PROGRAM DatenRangieren
VAR	
	VersionsText: STRING := 'LAP 2010/3 Ofentuersteuerung V3.0';
END_VAR

STRNCPY (ADR( _plcToPc.PlcToPc[96]), ADR( VersionsText), SIZEOF(VersionsText));

IF _PcToPlc.PcToPlc[96] = 16#00 THEN	// lokale Ein- und Ausgänge verwenden
	
ELSE	// Simulation (Digital Twin) verwenden
	
	_PlcToPc.PlcToPc[0] := AlleBitSetzen(	DA.P1,
											DA.Q1,
											DA.Q2,
											FALSE,	
											FALSE,	
											FALSE,	
											FALSE,										
											FALSE);	
											
	DI.B1 := BitLesen(_PcToPlc.PcToPlc[0],0);
	DI.B2 := BitLesen(_PcToPlc.PcToPlc[0],1);
	DI.B3 := BitLesen(_PcToPlc.PcToPlc[0],2);
	DI.S1 := BitLesen(_PcToPlc.PcToPlc[0],3);
	DI.S2 := BitLesen(_PcToPlc.PcToPlc[0],4);
	DI.S3 := BitLesen(_PcToPlc.PcToPlc[0],5);
END_IF

END_PROGRAM

(* stored: Version 1.1.0.1, ProductVersion 3.1.4024.5
   POU DatenRangieren: Id {ad49a684-d9e6-4dba-bece-08745f191ac1}, SpecialFunc None *)
